FUNCTION_BLOCK CmdDAerationValves (* CAT Function Block Type *)
  (* Standard: 61499-2 *)
  (* Version 0.0, 6/8/2026, Schneider Electric, template *)
  PACKAGE SE.Nereda;
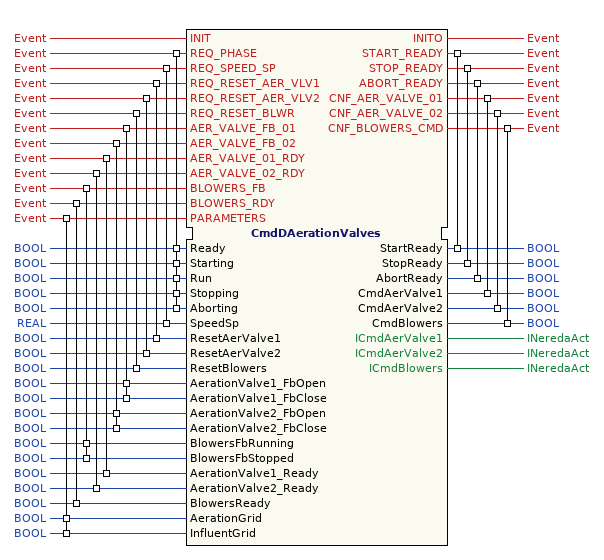
  EVENT_INPUT
    INIT;
    REQ_PHASE WITH Ready, Starting, Run, Stopping, Aborting;
    REQ_SPEED_SP WITH SpeedSp;
    REQ_RESET_AER_VLV1 WITH ResetAerValve1;
    REQ_RESET_AER_VLV2 WITH ResetAerValve2;
    REQ_RESET_BLWR WITH ResetBlowers;
    AER_VALVE_FB_01 WITH AerationValve1_FbOpen, AerationValve1_FbClose;
    AER_VALVE_FB_02 WITH AerationValve2_FbOpen, AerationValve2_FbClose;
    AER_VALVE_01_RDY WITH AerationValve1_Ready;
    AER_VALVE_02_RDY WITH AerationValve2_Ready;
    BLOWERS_FB WITH BlowersFbRunning, BlowersFbStopped;
    BLOWERS_RDY WITH BlowersReady;
    PARAMETERS WITH AerationGrid, InfluentGrid;
  END_EVENT
  EVENT_OUTPUT
    INITO;
    START_READY WITH StartReady;
    STOP_READY WITH StopReady;
    ABORT_READY WITH AbortReady;
    CNF_AER_VALVE_01 WITH CmdAerValve1;
    CNF_AER_VALVE_02 WITH CmdAerValve2;
    CNF_BLOWERS_CMD WITH CmdBlowers;
  END_EVENT
  VAR_INPUT
    Ready : BOOL;
    Starting : BOOL;
    Run : BOOL;
    Stopping : BOOL;
    Aborting : BOOL;
    SpeedSp : REAL;
    ResetAerValve1 : BOOL;
    ResetAerValve2 : BOOL;
    ResetBlowers : BOOL;
    AerationValve1_FbOpen : BOOL;
    AerationValve1_FbClose : BOOL;
    AerationValve2_FbOpen : BOOL;
    AerationValve2_FbClose : BOOL;
    BlowersFbRunning : BOOL;
    BlowersFbStopped : BOOL;
    AerationValve1_Ready : BOOL;
    AerationValve2_Ready : BOOL;
    BlowersReady : BOOL;
    AerationGrid : BOOL;
    InfluentGrid : BOOL;
  END_VAR
  VAR_OUTPUT
    StartReady : BOOL;
    StopReady : BOOL;
    AbortReady : BOOL;
    CmdAerValve1 : BOOL;
    CmdAerValve2 : BOOL;
    CmdBlowers : BOOL;
  END_VAR
  PLUGS
    ICmdAerValve1 : INeredaAct;
    ICmdAerValve2 : INeredaAct;
    ICmdBlowers : INeredaAct;
  END_PLUGS
  (* 01 - FUNCTIONNAL INPUT INTERFACE *)
  (* 00 - INITIALIZATION *)
  (* 05 - LOGIC *)
  (* 06 - HMI INTERFACE *)
  (* 03 - FIELD INTERFACE *)
  (* 02 - FUNCTIONNAL OUTPUT INTERFACE *)
  (* Command Logic *)
  FBS
    IThis : CmdDAerationValves_HMI(QI := TRUE);
    CmdLogic : CmdDAerationValvesBasic;
    CmdAerationValve1 : boolValueChanged;
    CmdAerationValve2 : boolValueChanged;
    CmdBlowersSmooth : boolValueChanged;
    FbOpenValve1 : DS_SELECTX_2536758B411A6CE51; {SET_ATTRIBUTE(Configuration.GenericFBType.InterfaceParams, Runtime.Standard#CNTX:=2;CNTY:=1;DI${CNTX,_,CNTY$}:BOOL)}
    FbCloseValve1 : DS_SELECTX_2536758B411A6CE51; {SET_ATTRIBUTE(Configuration.GenericFBType.InterfaceParams, Runtime.Standard#CNTX:=2;CNTY:=1;DI${CNTX,_,CNTY$}:BOOL)}
    FbRunBlowers : DS_SELECTX_2536758B411A6CE51; {SET_ATTRIBUTE(Configuration.GenericFBType.InterfaceParams, Runtime.Standard#CNTX:=2;CNTY:=1;DI${CNTX,_,CNTY$}:BOOL)}
    FbStopBlowers : DS_SELECTX_2536758B411A6CE51; {SET_ATTRIBUTE(Configuration.GenericFBType.InterfaceParams, Runtime.Standard#CNTX:=2;CNTY:=1;DI${CNTX,_,CNTY$}:BOOL)}
    FbReadyBlowers : DS_SELECTX_2536758B411A6CE51; {SET_ATTRIBUTE(Configuration.GenericFBType.InterfaceParams, Runtime.Standard#CNTX:=2;CNTY:=1;DI${CNTX,_,CNTY$}:BOOL)}
    FbReadyValve1 : DS_SELECTX_2536758B411A6CE51; {SET_ATTRIBUTE(Configuration.GenericFBType.InterfaceParams, Runtime.Standard#CNTX:=2;CNTY:=1;DI${CNTX,_,CNTY$}:BOOL)}
    FbOpenValve2 : DS_SELECTX_2536758B411A6CE51; {SET_ATTRIBUTE(Configuration.GenericFBType.InterfaceParams, Runtime.Standard#CNTX:=2;CNTY:=1;DI${CNTX,_,CNTY$}:BOOL)}
    FbCloseValve2 : DS_SELECTX_2536758B411A6CE51; {SET_ATTRIBUTE(Configuration.GenericFBType.InterfaceParams, Runtime.Standard#CNTX:=2;CNTY:=1;DI${CNTX,_,CNTY$}:BOOL)}
    FbReadyValve2 : DS_SELECTX_2536758B411A6CE51; {SET_ATTRIBUTE(Configuration.GenericFBType.InterfaceParams, Runtime.Standard#CNTX:=2;CNTY:=1;DI${CNTX,_,CNTY$}:BOOL)}
    Valve1Cmd : BOOL2INT;
    Valve2Cmd : BOOL2INT;
    BlowersCmd : BOOL2INT;
    RefreshParameters : E_CYCLE(DT := T#1s);
    CycleMng : StopStart;
  END_FBS
  EVENT_CONNECTIONS
    INIT TO IThis.3D5D26A512262747;
    IThis.5B84D78EC3FB5466 TO INITO;
    FbOpenValve1.CNF1 TO FbCloseValve1.REQ1;
    FbOpenValve1.CNF2 TO FbCloseValve1.REQ2;
    FbRunBlowers.CNF1 TO FbStopBlowers.REQ1;
    FbRunBlowers.CNF2 TO FbStopBlowers.REQ2;
    FbOpenValve2.CNF1 TO FbCloseValve2.REQ1;
    FbOpenValve2.CNF2 TO FbCloseValve2.REQ2;
    BLOWERS_RDY TO FbReadyBlowers.REQ2;
    BLOWERS_FB TO FbRunBlowers.REQ2;
    AER_VALVE_02_RDY TO FbReadyValve2.REQ2;
    AER_VALVE_01_RDY TO FbReadyValve1.REQ2;
    AER_VALVE_FB_02 TO FbOpenValve2.REQ2;
    AER_VALVE_FB_01 TO FbOpenValve1.REQ2;
    CmdLogic.2F06A37C5DC5770F TO IThis.FF79026EA8264D09;
    REQ_PHASE TO CmdLogic.0181C35002D51DB9;
    REQ_PHASE TO CmdLogic.7CF49D36E36F42BF;
    REQ_PHASE TO CmdLogic.270A548115E0D83C;
    REQ_PHASE TO CmdLogic.B01B36972B4703C3;
    REQ_PHASE TO CmdLogic.7D39C1849D7CD2AB;
    PARAMETERS TO CmdLogic.PARAMETERS;
    FbCloseValve1.IND TO CmdLogic.VALVE_036_FB_STATE;
    FbCloseValve2.IND TO CmdLogic.VALVE_067_FB_STATE;
    FbReadyValve1.IND TO CmdLogic.VALVE_036_AVAILABLE;
    FbReadyValve2.IND TO CmdLogic.VALVE_067_AVAILABLE;
    FbStopBlowers.IND TO CmdLogic.BLOWERS_STATE;
    FbReadyBlowers.IND TO CmdLogic.BLOWERS_NO_AVAILABLE;
    CmdLogic.CNF_VALVE_36 TO CmdAerationValve1.REQ;
    CmdLogic.CNF_VALVE_67 TO CmdAerationValve2.REQ;
    CmdLogic.CNF_BLOWERS TO CmdBlowersSmooth.REQ;
    CmdLogic.CNF_START_RDY TO START_READY;
    CmdLogic.CNF_STOP_RDY TO STOP_READY;
    CmdLogic.CNF_ABORT_RDY TO ABORT_READY;
    CmdAerationValve1.CHD TO Valve1Cmd.DD5870AA881150BB;
    CmdAerationValve2.CHD TO Valve2Cmd.DD5870AA881150BB;
    CmdBlowersSmooth.CHD TO BlowersCmd.DD5870AA881150BB;
    BlowersCmd.6FC99A5BD1C38561 TO CNF_BLOWERS_CMD;
    Valve2Cmd.6FC99A5BD1C38561 TO CNF_AER_VALVE_02;
    Valve1Cmd.6FC99A5BD1C38561 TO CNF_AER_VALVE_01;
    ICmdAerValve1.9CD053F8408797ED TO FbOpenValve1.REQ1;
    ICmdAerValve1.CC753684FA882790 TO FbReadyValve1.REQ1;
    ICmdAerValve2.9CD053F8408797ED TO FbOpenValve2.REQ1;
    ICmdAerValve2.CC753684FA882790 TO FbReadyValve2.REQ1;
    ICmdBlowers.9CD053F8408797ED TO FbRunBlowers.REQ1;
    ICmdBlowers.CC753684FA882790 TO FbReadyBlowers.REQ1;
    RefreshParameters.EO TO CmdLogic.PARAMETERS;
    CycleMng.36480E3E35BC8053 TO RefreshParameters.START;
    CycleMng.41BA9BA23CD04EBE TO RefreshParameters.STOP;
    REQ_PHASE TO CycleMng.9F78D3CDEE09DEB2;
  END_CONNECTIONS
  DATA_CONNECTIONS
    CmdBlowersSmooth.Output TO CmdBlowers;
    CmdAerationValve1.Output TO CmdAerValve1;
    CmdAerationValve2.Output TO CmdAerValve2;
    BlowersReady TO FbReadyBlowers.DI2_1;
    BlowersFbRunning TO FbRunBlowers.DI2_1;
    BlowersFbStopped TO FbStopBlowers.DI2_1;
    AerationValve2_Ready TO FbReadyValve2.DI2_1;
    AerationValve1_Ready TO FbReadyValve1.DI2_1;
    AerationValve2_FbClose TO FbCloseValve2.DI2_1;
    AerationValve2_FbOpen TO FbOpenValve2.DI2_1;
    AerationValve1_FbClose TO FbCloseValve1.DI2_1;
    AerationValve1_FbOpen TO FbOpenValve1.DI2_1;
    CmdLogic.CB6518449836B6D0 TO IThis.73E7435EE8FD8D21;
    Ready TO CmdLogic.Ready;
    Starting TO CmdLogic.Starting;
    Run TO CmdLogic.Run;
    Stopping TO CmdLogic.Stopping;
    Aborting TO CmdLogic.Aborting;
    SpeedSp TO ICmdBlowers.1BC103921BBFDA0B;
    ResetAerValve1 TO ICmdAerValve1.EA28053F07575F36;
    ResetAerValve2 TO ICmdAerValve2.EA28053F07575F36;
    ResetBlowers TO ICmdBlowers.EA28053F07575F36;
    AerationGrid TO CmdLogic.AerationGrid;
    InfluentGrid TO CmdLogic.InfluentGrid;
    FbOpenValve1.OUT1 TO CmdLogic.Valve036_FbOpen;
    FbCloseValve1.OUT1 TO CmdLogic.Valve036_FbClose;
    FbOpenValve2.OUT1 TO CmdLogic.Valve067_FbOpen;
    FbCloseValve2.OUT1 TO CmdLogic.Valve067_FbClose;
    FbReadyValve1.OUT1 TO CmdLogic.Valve036_Availabe;
    FbReadyValve2.OUT1 TO CmdLogic.Valve067_Availabe;
    FbRunBlowers.OUT1 TO CmdLogic.BlowersFbRunning;
    FbStopBlowers.OUT1 TO CmdLogic.BlowersFbStopped;
    FbReadyBlowers.OUT1 TO CmdLogic.BlowersNotAvailable;
    CmdLogic.Valve036 TO CmdAerationValve1.Input;
    CmdLogic.Valve067 TO CmdAerationValve2.Input;
    CmdLogic.Blowers TO CmdBlowersSmooth.Input;
    CmdLogic.StartReady TO StartReady;
    CmdLogic.StopReady TO StopReady;
    CmdLogic.AbortReady TO AbortReady;
    CmdAerationValve1.Output TO Valve1Cmd.4573FC8F228EB71D;
    CmdAerationValve2.Output TO Valve2Cmd.4573FC8F228EB71D;
    CmdBlowersSmooth.Output TO BlowersCmd.4573FC8F228EB71D;
    Valve1Cmd.A6DEF5F9C27C1848 TO ICmdAerValve1.710D7FC54EE3F35A;
    Valve2Cmd.A6DEF5F9C27C1848 TO ICmdAerValve2.710D7FC54EE3F35A;
    BlowersCmd.A6DEF5F9C27C1848 TO ICmdBlowers.710D7FC54EE3F35A;
    ICmdAerValve1.7F6CC7FEB9223DF3 TO FbOpenValve1.DI1_1;
    ICmdAerValve1.A8D6C4A1FDCCA991 TO FbCloseValve1.DI1_1;
    ICmdAerValve1.8A8A07EFCDA1443C TO FbReadyValve1.DI1_1;
    ICmdAerValve2.7F6CC7FEB9223DF3 TO FbOpenValve2.DI1_1;
    ICmdAerValve2.A8D6C4A1FDCCA991 TO FbCloseValve2.DI1_1;
    ICmdAerValve2.8A8A07EFCDA1443C TO FbReadyValve2.DI1_1;
    ICmdBlowers.D83B5BDEFA4D797C TO FbStopBlowers.DI1_1;
    ICmdBlowers.B762734C094A7162 TO FbRunBlowers.DI1_1;
    ICmdBlowers.8A8A07EFCDA1443C TO FbReadyBlowers.DI1_1;
    Run TO CycleMng.7E3D27FD59643C3E;
  END_CONNECTIONS
END_FUNCTION_BLOCK
